TYPE TcoSmartFunctionKitRequestHw_v_4_x_x : STRUCT
    Handle AT %Q* : WORD;
    Command AT %Q* : WORD;
    Value1 AT %Q* : DWORD;
    Value2 AT %Q* : DWORD;
    Value3 AT %Q* : DWORD;
    Value4 AT %Q* : DWORD;
    Value5 AT %Q* : DWORD;
    Value6 AT %Q* : DWORD;
    Value7 AT %Q* : DWORD;
    VirtualIo AT %Q* : WORD;
END_STRUCT
END_TYPE

(* stored: Version 1.1.0.1, ProductVersion 3.1.4024.11
   DUT TcoSmartFunctionKitRequestHw_v_4_x_x: Id {cd6bbd64-1cfc-0edb-06c9-2cb022502d39} *)
